(* CoDeSys 2.3 export: GETMV110INPUT.EXP *)

(* POU getMV110Input, ST *)
FUNCTION getMV110Input : BOOL
VAR_INPUT
	IN : USINT;
END_VAR
VAR
END_VAR
getMV110Input := EXTRACT(DI_1, IN);
END_FUNCTION
